FUNCTION f_mmToInch : REAL
VAR_INPUT
	rData : REAL;
END_VAR
VAR
END_VAR

f_mmToInch := rData * 0.0393701;

END_FUNCTION

(* stored: Version 1.1.0.1, ProductVersion 3.1.4024.12
   POU f_mmToInch: Id {d43840cb-667c-459a-bf74-8b26ff0757f5}, SpecialFunc None *)
